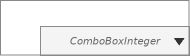
VISUALIZATION vTableFrameControl  // 190x56
VAR_IN_OUT
	fbTablePlace:FB_TablePlace;
END_VAR
    ComboBoxInteger (40,26 150x30), variable: fbTablePlace.stPlace.nState, text list: 'tlTableBottlePlaceState'
END_VISUALIZATION

(* stored: Version 1.1.0.1, ProductVersion 3.1.4024.15
   Visu vTableFrameControl: Id {bca8dcd2-0861-4c14-b458-c83274bb319c} *)
